// TwinCAT 3 PLC project Tests
// ProgramVersion: 3.1.4024.0
// libraries:
//   ADO_Demo_PLC, * (Beckhoff)
//   Tc2_Standard, * (Beckhoff Automation GmbH)
//   Tc2_System, * (Beckhoff Automation GmbH)
//   Tc3_Module, * (Beckhoff Automation GmbH)
//   TcUnit, * (www.tcunit.org)
// project tree:
//   / PlcTask.TcTTO
//   Test/ FB_CellCheckPart_Test.TcPOU, PRG_TEST.TcPOU
// (motion and I/O tree: see PLC project plc)
// real-time tasks:
//   TASK PlcTask: cycle T#10ms, priority 20, ADS port 350
//   TASK PlcTask1: cycle T#10ms, priority 21, ADS port 351
// variable links:

CONFIGURATION Tests
    RESOURCE PLC ON TwinCAT3
        TASK PlcTask(INTERVAL := T#10ms, PRIORITY := 21);
        PROGRAM PRG_TEST WITH PlcTask : PRG_TEST;
    END_RESOURCE
END_CONFIGURATION

// ---- Test/PRG_TEST.TcPOU
PROGRAM PRG_TEST
VAR
	fbCheckPartTest		: FB_CellCheckPart_Test;
END_VAR

TcUnit.RUN();

END_PROGRAM

// ---- Test/FB_CellCheckPart_Test.TcPOU
FUNCTION_BLOCK FB_CellCheckPart_Test EXTENDS TcUnit.FB_TestSuite
VAR
END_VAR

CheckPartGood();
CheckPartBadBarcode();

METHOD PRIVATE CheckPartBadBarcode
VAR
	fbCell		: ADO_Demo_PLC.FB_Cell;
	MockStatus	: ADO_Demo_PLC.ST_PartStatus;
	Expected	: BOOL := FALSE;
	Result		: BOOL;
END_VAR
MockStatus.bBarcodeStatus := FALSE;
MockStatus.bCapperStatus := TRUE;
MockStatus.bFillerStatus := TRUE;
MockStatus.bWeightStatus := TRUE;

Result := fbCell.CheckPart(MockStatus);

AssertEquals(Expected := Expected,
             Actual := Result,
             Message := 'part check mismatch');

TEST_FINISHED();
END_METHOD

METHOD PRIVATE CheckPartGood
VAR
	fbCell		: ADO_Demo_PLC.FB_Cell;
	MockStatus	: ADO_Demo_PLC.ST_PartStatus;
	Expected	: BOOL := TRUE;
	Result		: BOOL;
END_VAR
MockStatus.bBarcodeStatus := TRUE;
MockStatus.bCapperStatus := TRUE;
MockStatus.bFillerStatus := TRUE;
MockStatus.bWeightStatus := TRUE;

Result := fbCell.CheckPart(MockStatus);

AssertEquals(Expected := Expected,
             Actual := Result,
             Message := 'part check mismatch');

TEST_FINISHED();
END_METHOD

END_FUNCTION_BLOCK
